{attribute wpf [Container(Layout.Wrap)]}
{attribute wpf [Group(Layout.GroupBox)]}
FUNCTION_BLOCK fbStepConveyor
VAR_INPUT
	{attribute wpf [Container(Layout.Stack)]}	
	{attribute addProperty Name "Stop condition"}
	{attribute addProperty ToolTip "Signal that stops the conveyor"}
	inStop : BOOL;	
END_VAR
VAR_OUTPUT
	{attribute wpf [Container(Layout.Stack)]}
	{attribute addProperty Name "Move"}
	{attribute addProperty ToolTip "Signal for moving conveyor"}
	outMove : BOOL;
END_VAR
VAR
	{attribute wpf [Container(Layout.UniformGrid)]}
	{attribute addProperty Name "Move manual command"}
	{attribute addProperty ToolTip "Triggers movement in manual mode if possible"}
	_manualMove : BOOL;	
	{attribute 'hide'}
	_move : BOOL;	
	{attribute 'hide'}
	rtrg_inStop : R_TRIG;	
	{attribute 'hide'}
	_moveTimeout : TON;	
END_VAR

rtrg_inStop(CLK := inStop);

_moveTimeout(IN := THIS^._move, PT := T#500MS);

IF rtrg_inStop.Q OR _moveTimeout.Q THEN
	_move := FALSE;
END_IF


THIS^.outMove := _move;

METHOD Manual
IF THIS^._manualMove THEN THIS^._move := TRUE; END_IF;

THIS^._manualMove := FALSE;
END_METHOD

PROPERTY Run : BOOL
GET
END_GET
SET
_move := RUN;
END_SET
END_PROPERTY

END_FUNCTION_BLOCK

(* stored: Version 1.1.0.1, ProductVersion 3.1.4024.2
   POU fbStepConveyor: Id {7e0f4cfc-9cb7-42de-b49f-70bfef52e2b0}, SpecialFunc None
   Method Manual: Id {c189c067-fde9-444b-aad0-5e7ebd281a50}
   Property Run: Id {b4822184-83ee-442b-bef3-e48e30621107}
   Get Get: Id {6d7fd730-2ef9-4833-85cb-83e91c3066ef}
   Set Set: Id {8f284d37-d2bd-4a50-aef3-1e205ee092e9} *)
